TYPE ST_OutputCellAdditionalData :
STRUCT
	{attribute 'OPC.UA.DA.Description' := 'Dummy (for making struct visible on OPC UA'}
	Dummy						: BOOL;

END_STRUCT
END_TYPE

(* stored: Version 1.1.0.1, ProductVersion 3.1.4024.2
   DUT ST_OutputCellAdditionalData: Id {ebe76aab-9688-440d-af5c-fa51866bb041} *)
